// ---- 32_UML_StateChart/32_VISU/_32_Visualization.TcVIS
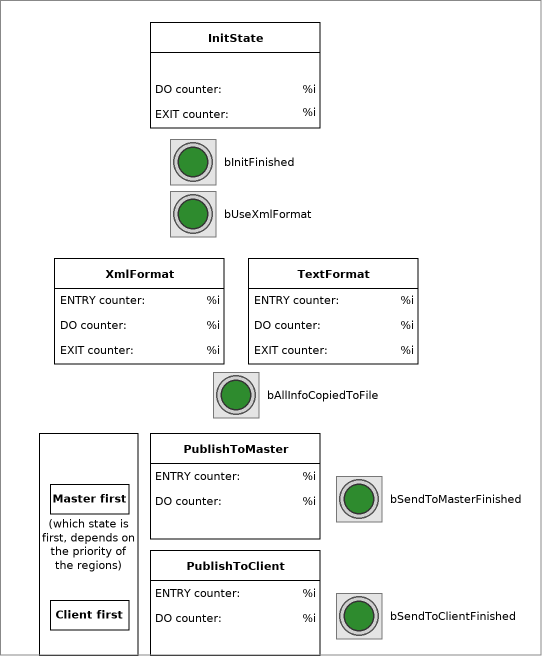
VISUALIZATION _32_Visualization  // 542x656
    Rectangle (39,433 99x223), "(which state is first, depends on the priority of the regions)"
    Rectangle (150,22 170x106)
    Label (152,27 168x23), "InitState"
    Rectangle (54,258 170x106)
    Label (56,263 168x23), "XmlFormat"
    Rectangle (248,258 170x106)
    Label (250,263 168x23), "TextFormat"
    Rectangle (150,433 170x106)
    Label (152,438 168x23), "PublishToMaster"
    Rectangle (150,550 170x106)
    Label (152,555 168x23), "PublishToClient"
    PushSwitch (170,139 46x46), variable: _32_MAIN.fbUmlSC.bInitFinished, behaviour: TOGGLE, style: Switch-PushSwitch-Green
    Label (221,151 118x23), "bInitFinished"
    PushSwitch (170,191 46x46), variable: _32_MAIN.fbUmlSC.bUseXmlFormat, behaviour: TOGGLE, style: Switch-PushSwitch-Green
    Label (221,203 118x23), "bUseXmlFormat"
    PushSwitch (213,372 46x46), variable: _32_MAIN.fbUmlSC.bAllInfoCopiedToFile, behaviour: TOGGLE, style: Switch-PushSwitch-Green
    Label (264,384 137x23), "bAllInfoCopiedToFile"
    PushSwitch (336,476 46x46), variable: _32_MAIN.fbUmlSC.bSendToMasterFinished, behaviour: TOGGLE, style: Switch-PushSwitch-Green
    Label (387,488 155x23), "bSendToMasterFinished"
    PushSwitch (336,593 46x46), variable: _32_MAIN.fbUmlSC.bSendToClientFinished, behaviour: TOGGLE, style: Switch-PushSwitch-Green
    Label (387,605 141x23), "bSendToClientFinished"
    Rectangle (152,79 90x21), "DO counter:", text variable: _32_MAIN.fbUmlSC.nCounterInit
    Rectangle (152,104 90x21), "EXIT counter:", text variable: _32_MAIN.fbUmlSC.nCounterSaveInitSettings
    Rectangle (57,290 90x21), "ENTRY counter:", text variable: _32_MAIN.fbUmlSC.nCounterClearXml
    Rectangle (57,315 90x21), "DO counter:", text variable: _32_MAIN.fbUmlSC.nCounterFillXml
    Rectangle (57,340 90x21), "EXIT counter:", text variable: _32_MAIN.fbUmlSC.nCounterSaveXml
    Rectangle (251,290 90x21), "ENTRY counter:", text variable: _32_MAIN.fbUmlSC.nCounterClearText
    Rectangle (251,315 90x21), "DO counter:", text variable: _32_MAIN.fbUmlSC.nCounterFillText
    Rectangle (251,340 90x21), "EXIT counter:", text variable: _32_MAIN.fbUmlSC.nCounterSaveText
    Rectangle (152,466 90x21), "ENTRY counter:", text variable: _32_MAIN.fbUmlSC.nCounterGetMasterID
    Rectangle (152,491 90x21), "DO counter:", text variable: _32_MAIN.fbUmlSC.nCounterSendToMaster
    Rectangle (152,583 90x21), "ENTRY counter:", text variable: _32_MAIN.fbUmlSC.nCounterGetClientID
    Rectangle (152,608 90x21), "DO counter:", text variable: _32_MAIN.fbUmlSC.nCounterSendToClient
    Line (150,52) (320,52)
    Line (248,288) (418,288)
    Line (54,288) (224,288)
    Line (150,463) (320,463)
    Line (150,580) (320,580)
    Rectangle (249,79 70x21), "%i", text variable: _32_MAIN.fbUmlSC.nCounterInit
    Rectangle (249,102 70x21), "%i", text variable: _32_MAIN.fbUmlSC.nCounterSaveInitSettings
    Rectangle (153,290 70x21), "%i", text variable: _32_MAIN.fbUmlSC.nCounterClearXml
    Rectangle (153,315 70x21), "%i", text variable: _32_MAIN.fbUmlSC.nCounterFillXml
    Rectangle (153,340 70x21), "%i", text variable: _32_MAIN.fbUmlSC.nCounterSaveXml
    Rectangle (347,290 70x21), "%i", text variable: _32_MAIN.fbUmlSC.nCounterClearText
    Rectangle (347,315 70x21), "%i", text variable: _32_MAIN.fbUmlSC.nCounterFillText
    Rectangle (347,340 70x21), "%i", text variable: _32_MAIN.fbUmlSC.nCounterSaveText
    Rectangle (249,466 70x21), "%i", text variable: _32_MAIN.fbUmlSC.nCounterGetMasterID
    Rectangle (249,491 70x21), "%i", text variable: _32_MAIN.fbUmlSC.nCounterSendToMaster
    Rectangle (249,583 70x21), "%i", text variable: _32_MAIN.fbUmlSC.nCounterGetClientID
    Rectangle (249,608 70x21), "%i", text variable: _32_MAIN.fbUmlSC.nCounterSendToClient
    Rectangle (50,484 79x30), "Master first", colour toggle: _32_MAIN.fbUmlSC.bMasterFirst
    Rectangle (50,600 79x30), "Client first", colour toggle: _32_MAIN.fbUmlSC.bClientFirst
END_VISUALIZATION

// ---- GlobalTextList.TcGTLO
TEXTLIST GlobalTextList
  414 = '\n(which state is first, depends on the priority of the regions)'
  160 = '%i'
  10 = 'bAllInfoCopiedToFile'
  8 = 'bInitFinished'
  12 = 'bSendToClientFinished'
  11 = 'bSendToMasterFinished'
  9 = 'bUseXmlFormat'
  241 = 'Client first'
  332 = 'DO counter:'
  846 = 'ENTRY counter:'
  807 = 'EXIT counter:'
  3 = 'InitState'
  197 = 'Master first'
  7 = 'PublishToClient'
  6 = 'PublishToMaster'
  5 = 'TextFormat'
  4 = 'XmlFormat'
END_TEXTLIST
